FUNCTION_BLOCK AppContext EXTENDS TcoCore.TcoContext
VAR
    _mainStation : MainStation(THIS^);

    {attribute addProperty Name "Versionsnummer Plc"}
    _sVersion : STRING(23);
    //~
    _stProgramVersion : ST_LibVersion;
    //~

END_VAR

(*~
    <docu>
        <summary>
            Main method of the TcoContext. This is the entry point of any control logic that belongs to this context.
            The call of this method is ensured by calling the <c>InstanceName.Run()</c> method, and it must not be called explicitly.
            This method is abstract, and it must be overridden in derived block.
        </summary>
    </docu>
~*)
METHOD PROTECTED Main
_mainStation();

//IF (THIS^._startCycleCount MOD 10 = 0) THEN
//    Logger.Push('This is a log entry', eMessageCategory.Trace);
//END_IF;

//IF (THIS^._startCycleCount MOD 125 = 0) THEN
//    Logger.Push('This is a log entry', eMessageCategory.Info);
//END_IF;

//IF (THIS^._startCycleCount MOD 400 = 0) THEN
//    Logger.Push('This is a log entry', eMessageCategory.Warning);
//END_IF;

//IF (THIS^._startCycleCount MOD 2000 = 0) THEN
//    Logger.Push('This is a log entry', eMessageCategory.Error);
//END_IF;
END_METHOD

END_FUNCTION_BLOCK

(* stored: Version 1.1.0.1, ProductVersion 3.1.4024.12
   POU AppContext: Id {13bf0f33-380e-0bed-2b6e-cf8581b41dee}, SpecialFunc None
   Method Main: Id {e0bc1bc7-e259-0efa-2e7d-4ebd073a0fbb} *)
